(* IEC 61131-3 sources: inproshop/test13_exported/OP20/2.PRG, 9 files *)

(* ---- OP20_Communication.st ---- *)
PROGRAM OP20_Communication
VAR
	HeartdelayON:TON;
	HeartdelayOFF:TON;
	MasterHeartdelayON:TON;
	MasterHeartdelayOFF:TON;
END_VAR

//心跳输出
IF CPU_Clock.Clock_1s THEN
	DB2005_Communication.TO_OPXX.Heart:=1;
ELSE
	DB2005_Communication.TO_OPXX.Heart:=0;
END_IF
//给前站安全信号
IF TRUE THEN
	DB2005_Communication.TO_OPXX.Safe:=1;
ELSE
	DB2005_Communication.TO_OPXX.Safe:=0;
END_IF;

HeartdelayON(IN:= DB2005_Communication.From_OPXX.Heart=1, PT:= T#2S, Q=> , ET=> );
HeartdelayOFF(IN:= DB2005_Communication.From_OPXX.Heart=0, PT:= T#2S, Q=> , ET=> );
//前站掉线报警
IF (HeartdelayON.Q OR HeartdelayOFF.Q) AND NOT DB2000_Control.Mode.Status.OfflineMode  THEN
	DB2070_Fault.Stop.BeforStation_Communication_Rrror:=TRUE;
END_IF

//主站心跳通讯检测
MasterHeartdelayON(IN:= DB2005_Communication.FromMaster.Heart=1, PT:= T#2S, Q=> , ET=> );
MasterHeartdelayOFF(IN:= DB2005_Communication.FromMaster.Heart=0, PT:= T#2S, Q=> , ET=> );
//主站掉线报警
IF (MasterHeartdelayON.Q OR MasterHeartdelayOFF.Q) AND NOT DB2000_Control.Mode.Status.OfflineMode  THEN
	DB2070_Fault.Stop.MasterTimeOut:=TRUE;
END_IF

//与主站配方不一致报警
IF DB2005_Communication.FromMaster.MasterRecipeID<>DB2002_Recipe.RecipeNum AND NOT DB2000_Control.Mode.Status.OfflineMode THEN
	DB2070_Fault.Stop.MaterReipeDiscrepancy:=TRUE;
END_IF

(* ---- OP20_Control.st ---- *)
PROGRAM OP20_Control
VAR
	FB_ModeControl_instance:FB_ModeControl_V1;
	FB_Count_instance:ARRAY[0..2] OF FB_Count;
END_VAR

(**********模式切换功能***********)
FB_ModeControl_instance(
	iClock:= CPU_Clock,
	iStartDelay:= T#100MS,
	iEstop:=DB2070_Fault.EstopTotal,
	iAlam:=DB2070_Fault.StopTotal,
	iWarn:=DB2070_Fault.RunTotal,
	ioMachine:= DB2000_Control.Machine,
	ioMode:=DB2000_Control.Mode);

(********************计数****************************)
//总计数
FB_Count_instance[0](
	ioCount:= DB2003_Count.Total,
	iClock:= CPU_Clock,
	iDayStartTime:= CPU_Clock.DayStartTime,
	iNightStartTime:=CPU_Clock.NightStartTime);

//OK计数
FB_Count_instance[1](
	ioCount:= DB2003_Count.OK,
	iClock:= CPU_Clock,
	iDayStartTime:= CPU_Clock.DayStartTime,
	iNightStartTime:=CPU_Clock.NightStartTime);

//NG计数
FB_Count_instance[2](
	ioCount:= DB2003_Count.NG,
	iClock:= CPU_Clock,
	iDayStartTime:= CPU_Clock.DayStartTime,
	iNightStartTime:=CPU_Clock.NightStartTime);

(***********良率计算***********)
//良率统计
IF DB2003_Count.Total.Today.Total<>0 THEN
	DB2003_Count.Yield:=DB2003_Count.OK.Today.Total/DB2003_Count.Total.Today.Total;
ELSE
	DB2003_Count.Yield:=0;
END_IF
//良率清零
IF DB2003_Count.Clear THEN
	DB2003_Count.Total.Today.Total:=0;
	DB2003_Count.OK.Today.Total:=0;
	DB2003_Count.NG.Today.Total:=0;
	DB2003_Count.Clear:=FALSE;
END_IF

(********程序调用*******)
OP20_DI_Mirror();
OP20_Communication();
OP20_Recipe();
OP20_Graph();
OP20_DriveControl();
OP20_DO_Mirror();
OP20_Fault();
OP20_Other();

(* ---- OP20_DI_Mirror.st ---- *)
PROGRAM OP20_DI_Mirror
VAR
	i:INT;//循环用变量
	Page:INT;
	Monitor:ARRAY[0..15] OF Str_IOMonitor;
	Status:WORD;
	Map:BOOL;
END_VAR

ACT_MAP();
ACT_Comment();
ACT_Status();

(* ---- OP20_DO_Mirror.st ---- *)
PROGRAM OP20_DO_Mirror
VAR
	i:INT;//循环用变量
	Page:INT;
	Monitor:ARRAY[0..15] OF Str_IOMonitor;
	Status:WORD;
	Map:BOOL;
	Startlamp1:BOOL;
	Startlamp2:BOOL;
END_VAR

ACT_MAP();
ACT_Comment();
ACT_Status();

(* ---- OP20_DriveControl.st ---- *)
PROGRAM OP20_DriveControl
VAR
	FB_Cylinder_instance :ARRAY[0..63]OF FB_Cylinder_V1;
	FB_Vacuum_instance :ARRAY[0..31]OF FB_Vacuum_V1;
	FB_Axis_Instance:ARRAY[0..31]OF FB_Axis_V1_3;
	FB_Sensor_instance :ARRAY[0..200]OF FB_Sensor_V1_1;
	FB_TcpClient_Instance:ARRAY[0..31]OF FB_TcpClient;
	FB_DoubleStart_Instance:ARRAY[1..4]OF FB_DoubleStart;
	FB_Epson_V1_Instance:ARRAY[1..1]OF FB_Epson_V1;
	FB_Kuka_V1_Instance:ARRAY[1..2]OF FB_Kuka6_V1;
	FB_Rotdisk_V1_Instance:ARRAY[1..1]OF FB_Rotdisk_V1;
	FB_Stopper_V1_Instance:ARRAY[1..1]OF FB_Stopper_V1;
	FB_Motor_Instance:ARRAY[1..1]OF FB_Motor;
	FB_Heating_Instance:ARRAY[1..1]OF FB_Heating;
	FB_Gear_Instance:ARRAY[1..1]OF FB_Gear;
	FB_AAS_Instance:ARRAY[1..1]OF FB_AAS;
	FB_AirLeak_Instance:ARRAY[1..2]OF FB_AirLeak;
	FB_Palletizing_Instance:ARRAY[1..3]OF FB_Palletizing;
END_VAR
VAR
	i:INT;//循环变量用
	j:INT;//循环变量用
END_VAR

VAR
	TempKUKA1InPut AT %IB4500:ARRAY[0..63]OF BYTE;
	TempKUKA1OutPut AT %QB4500:ARRAY[0..63]OF BYTE;
	TempKUKA2InPut AT %IB4600:ARRAY[0..63]OF BYTE;
	TempKUKA2OutPut AT %QB4600:ARRAY[0..63]OF BYTE;
END_VAR
VAR
	PowerLimitDelay:ARRAY[0..16] OF TON;//超出额定电流
END_VAR

ACT_Axis();
ACT_Cylinder();
ACT_Vacuum();
ACT_Epson();
ACT_Kuka();
ACT_Sensor();
ACT_Motor();
ACT_Rotdisk();
ACT_AI();
ACT_Stopper();

ACT_Pallet();

(* ---- OP20_Fault.st ---- *)
PROGRAM OP20_Fault
VAR
	i:UINT;//循环变量用
	Pobool_IN: POINTER TO BOOL;//输入报警指针地址获取；
	Pobool_OUT: POINTER TO BOOL;//输出报警指针地址获取；
	EstopMAP:ARRAY[0..255] OF BOOL;
	StopMAP:ARRAY[0..999] OF BOOL;
	RunMAP:ARRAY[0..255] OF BOOL;
	Size:UINT;//数组数量
	Estop_R:R_TRIG;//急停上升沿
	Stop_R:R_TRIG;//暂停上升沿
	Run_R:R_TRIG;//警告上升沿
	StopFaultDelay:ARRAY[1..10]OF TON;//停止报警延时
END_VAR

//气缸报警地址映射
SizeOfAry(In:=DB2050_DriveControl.CylCtrl,Out=>Size);
FOR i:=0 TO Size-1 BY 1 DO
	DB2070_Fault.Stop.Cyl[I]:=DB2050_DriveControl.CylCtrl[i].Status.Error;
END_FOR
//真空报警映射
SizeOfAry(In:=DB2050_DriveControl.VacCtrl,Out=>Size);
FOR i:=0 TO Size-1 BY 1 DO
	DB2070_Fault.Stop.Vac[I]:=DB2050_DriveControl.VacCtrl[i].Status.Error;
END_FOR
//轴报警映射
SizeOfAry(In:=DB2050_DriveControl.AxisCtrl,Out=>Size);
FOR i:=0 TO Size-1 BY 1 DO
	DB2070_Fault.Stop.Axis[I]:=DB2050_DriveControl.AxisCtrl[i].Status.Error;
END_FOR

//急停报警
DB2070_Fault.Estop.EstopButton:=NOT DB2000_Control.Machine.EmgSafetyRelay;

//暂停故障

//提示

ACT_MAP();
ACT_HMI_Jump();

(* ---- OP20_Graph.st ---- *)
PROGRAM OP20_Graph
VAR
	IntitalTimeDelay:ARRAY[1..9,0..10] OF TON;//初始化流程用
	AutoTimeDelay:ARRAY[1..9,0..10] OF TON;//自动流程用

	Init:ARRAY[1..20]OF Str_Graph := [20((Complete := TRUE))];//初始化
	Auto:ARRAY[1..20]OF Str_Graph;//自动
	Start:ARRAY[1..9] OF BOOL;//自动启动条件
	i:INT;//循环变量用

	AgingPutAllowNo:INT;//老化允许放编号
	AgingPickAllowNo:INT;//老化允许取编号
	BufferPutAllowNo:INT;//缓存台允许放编号

	AgingPutAllow:BOOL;//老化允许放
	AgingPickAllow:BOOL;//老化允许取
	BufferPutAllow:BOOL;//缓存台允许放

	BufferPickAllow:BOOL;//缓存台允许取
	TestPickAllow:BOOL;//测试台允许取
	TestPutAllow:BOOL;//测试台允许放
	PalletProductPutAllow:BOOL;//码垛区域允许放产品
	PalletPartitionPutAllow:BOOL;//码垛区域允许放隔板
	PalletPartitionPickAllow:BOOL;//码垛区域允许取隔板
	NgPutAllow:BOOL;//NG区域允许放料

	BufferPickAllowNo:INT;//缓存台允许取编号
	TestPickAllowNo:INT;//测试台允许取编号
	TestPutAllowNo:INT;//测试台允许放编号
	PalletProductPutAllowNo:INT;//码垛区域允许放产品编号
	PalletPartitionPutAllowNo:INT;//码垛区域允许放隔板编号

	PartitionInRobot:BOOL;//机械手上有隔板

	X1Point:INT;//X1轴
	X2Point:INT;//X1轴
	BufferDisable:ARRAY[0..4]OF BOOL;

END_VAR

ACT_InitST1();
ACT_InitST2();
ACT_InitST3();
ACT_InitST4();
ACT_InitST5();
ACT_InitST6();

ACT_AutoRunST1_气密1测试();
ACT_AutoRunST2_气密2测试();
ACT_AutoRunST3_气密3测试();
ACT_AutoRunST4_气密4测试();
ACT_AutoRunST5_上料机械手();
ACT_AutoRunST6_码垛机械手();

(* ---- OP20_Other.st ---- *)
PROGRAM OP20_Other
VAR
	i:INT;//循环变量
	MaterialCode: INT;
END_VAR

(* ---- OP20_Recipe.st ---- *)
PROGRAM OP20_Recipe
VAR
	i:INT;
	DownLoad_R:R_TRIG;
	Download_F:F_TRIG;
	Change:R_TRIG;
END_VAR
VAR RETAIN PERSISTENT
	RecipeNum AT %MB131076 : INT;
END_VAR

//主站一键切换配方
IF To_Slave.OnLineMode=1 THEN
	IF DB2002_Recipe.DownLoad THEN
		To_Slave.RecipeDownLoad:=1;
	ELSE
		To_Slave.RecipeDownLoad:=0;
	END_IF
	To_Slave.RecipeID:=DB2002_Recipe.RecipeNumTemp;
ELSE
	To_Slave.RecipeDownLoad:=0;
END_IF

//配方名
DB2002_Recipe.RecipeName:=DB2002_Recipe.TypeData[DB2002_Recipe.RecipeNum].Name;

//配方参数修改使能
IF DB2002_Recipe.RecipeNum=DB2002_Recipe.RecipeNumTemp THEN
	DB2002_Recipe.ParameterChangePmt:=TRUE;
ELSE
	DB2002_Recipe.ParameterChangePmt:=FALSE;
END_IF

//配方允许切换使能
DB2002_Recipe.RecipeChangePmt:=DB2000_Control.Mode.Status.ManualMode ;

//配方提取
DB2002_Recipe.TypeDataCur:=DB2002_Recipe.TypeData[DB2002_Recipe.RecipeNum];

IF RecipeNum<>DB2002_Recipe.RecipeNumTemp THEN
	DB2002_Recipe.RecipeNameTemp:=DB2002_Recipe.TypeData[DB2002_Recipe.RecipeNumTemp].Name;
	RecipeNum:=DB2002_Recipe.RecipeNumTemp;
END_IF

DownLoad_R(CLK:= DB2002_Recipe.DownLoad);
DownLoad_F(CLK:= DB2002_Recipe.DownLoad);
ACT_Download();
ACT_Upload();
